{attribute 'qualified_only'}

TYPE eColorOrder :
(
	RGB := 0,
	GRB := 1
);
END_TYPE

(* stored: Version 1.1.0.1, ProductVersion 3.1.4026.18
   DUT eColorOrder: Id {910bcf7c-8135-4a04-a17c-265e6256987c} *)
